// TIA Portal project "烧嘴报警程序" (V17)

(* hardware
DEVICE "PLC_1"  S7-1200 Station
   slot 0: "Rack_0"  S7-1200 Rack  Rack  V1.0
   slot 1: "PLC_1"  CPU 1214C DC/DC/DC  6ES7 214-1AG40-0XB0  V4.5
*)

// ===== PLC "PLC_1"  CPU 1214C DC/DC/DC =====

VAR_GLOBAL   // PLC tag table "烧嘴报警变量"
   "1#故障反馈" AT %I0.1 : Bool;
   "2#故障反馈" AT %I0.4 : Bool;
   "3#故障反馈" AT %I0.7 : Bool;
   "4#故障反馈" AT %I1.2 : Bool;
   "5#故障反馈" AT %I1.5 : Bool;
   "6#故障反馈" AT %I2.2 : Bool;
   "7#故障反馈" AT %I2.5 : Bool;
   "蜂鸣器" AT %Q4.7 : Bool;
END_VAR

DATA_BLOCK "内部数据"   // DB1
{ S7_Optimized_Access := 'TRUE' }
VERSION : 0.1
   VAR
      报警脉冲 : Bool;   // 故障报警脉冲存储
      控温超温标志 : Bool;   // 控温超温汇总标志
   END_VAR
BEGIN
END_DATA_BLOCK

DATA_BLOCK "数字量信号"   // DB2
{ S7_Optimized_Access := 'TRUE' }
VERSION : 0.1
   VAR
      _1区超温标志 : Bool;   // 1区超温标志
      _2区超温标志 : Bool;   // 2区超温标志
      _3区超温标志 : Bool;   // 3区超温标志
      _4区超温标志 : Bool;   // 4区超温标志
      _5区超温标志 : Bool;   // 5区超温标志
      _6区超温标志 : Bool;   // 6区超温标志
   END_VAR
BEGIN
END_DATA_BLOCK

FUNCTION "FC_烧嘴报警" : Void   // FC1, LAD
{ S7_Optimized_Access := 'TRUE' }
   VAR_TEMP   // added for the SCL form of the ladder/FBD networks
      _w1 : Bool;
      _w2 : Bool;
   END_VAR
BEGIN

REGION Network 1: 故障反馈汇总与蜂鸣器报警
   // 任意烧嘴故障反馈上升沿时置位蜂鸣器输出
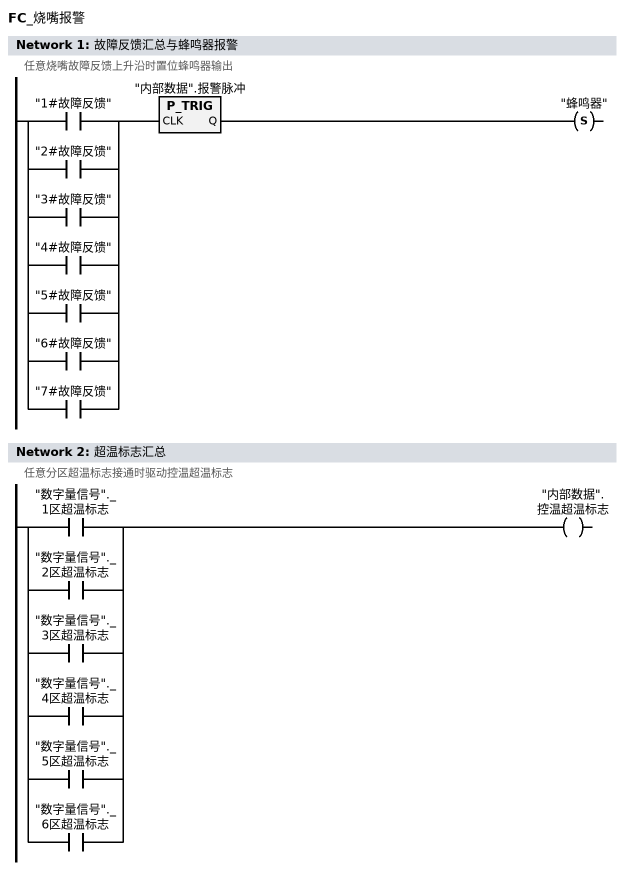
   RUNG wire#powerrail
      Contact( "1#故障反馈" )
      wire#w1
      P_Trig( "内部数据".报警脉冲 )
      S_Coil( "蜂鸣器" )
   END_RUNG
   RUNG wire#powerrail
      Contact( "2#故障反馈" )
   END_RUNG wire#w1
   RUNG wire#powerrail
      Contact( "3#故障反馈" )
   END_RUNG wire#w1
   RUNG wire#powerrail
      Contact( "4#故障反馈" )
   END_RUNG wire#w1
   RUNG wire#powerrail
      Contact( "5#故障反馈" )
   END_RUNG wire#w1
   RUNG wire#powerrail
      Contact( "6#故障反馈" )
   END_RUNG wire#w1
   RUNG wire#powerrail
      Contact( "7#故障反馈" )
   END_RUNG wire#w1
   // the same network as SCL:
   #_w1 := "1#故障反馈" OR "2#故障反馈" OR "3#故障反馈" OR "4#故障反馈" OR "5#故障反馈" OR "6#故障反馈" OR "7#故障反馈";
   #_w2 := #_w1 AND NOT "内部数据".报警脉冲;   // rising edge
   "内部数据".报警脉冲 := #_w1;
   IF #_w2 THEN "蜂鸣器" := TRUE; END_IF;
END_REGION

REGION Network 2: 超温标志汇总
   // 任意分区超温标志接通时驱动控温超温标志
   RUNG wire#powerrail
      Contact( "数字量信号"._1区超温标志 )
      wire#w1
      Coil( "内部数据".控温超温标志 )
   END_RUNG
   RUNG wire#powerrail
      Contact( "数字量信号"._2区超温标志 )
   END_RUNG wire#w1
   RUNG wire#powerrail
      Contact( "数字量信号"._3区超温标志 )
   END_RUNG wire#w1
   RUNG wire#powerrail
      Contact( "数字量信号"._4区超温标志 )
   END_RUNG wire#w1
   RUNG wire#powerrail
      Contact( "数字量信号"._5区超温标志 )
   END_RUNG wire#w1
   RUNG wire#powerrail
      Contact( "数字量信号"._6区超温标志 )
   END_RUNG wire#w1
   // the same network as SCL:
   "内部数据".控温超温标志 := "数字量信号"._1区超温标志 OR "数字量信号"._2区超温标志 OR "数字量信号"._3区超温标志 OR "数字量信号"._4区超温标志 OR "数字量信号"._5区超温标志 OR "数字量信号"._6区超温标志;
END_REGION
END_FUNCTION

ORGANIZATION_BLOCK "Main"   // OB1, LAD, ProgramCycle
TITLE = "Main Program Sweep (Cycle)"
{ S7_Optimized_Access := 'TRUE' }
VERSION : 0.1
   VAR_INPUT
      Initial_Call : Bool;   // Initial call of this OB
      Remanence : Bool;   // =True, if remanent data are available
   END_VAR
BEGIN
END_ORGANIZATION_BLOCK